// SIMATIC STEP 7 (V5.x) project GRAFCET__DELAY

SYMBOL_TABLE
"Motor Program"	FB 1	FB 1
"G7_STD_3"	FC 72	FC 72
"Start Btn"	I 0.0	BOOL	// Start cycle button input
"Reset Btn"	I 0.1	BOOL	// Reset cycle button input
"Cycle Execution"	OB 1	OB 1
"KM"	Q 0.0	BOOL	// Output motor to drive
"TIME_TCK"	SFC 64	SFC 64	// Read the System Time
END_SYMBOL_TABLE
